{attribute 'GeneratedUsingTerminal: EL6631-0000-0018'}
{attribute addProperty BoxType "EL6631-0000-0018"}
{attribute addProperty Id "AdsAddrAT %I*TcoIo.TcoAmsAddr0AoeNetIdAT %I*TcoIo.TcoAmsNetId0StateAT %I*UINT2"}
{attribute addProperty CRC "2407881067"}
{attribute addProperty Size "2"}
TYPE InfoData_8F85596B EXTENDS TcoIo.InputBase_8311D824 :
STRUCT
	{attribute addProperty Name "AdsAddr"}
	AdsAddr AT %I* : TcoIo.TcoAmsAddr;
	{attribute addProperty Name "AoeNetId"}
	AoeNetId AT %I* : TcoIo.TcoAmsNetId;
	{attribute addProperty Name "State"}
	State AT %I* : UINT;
END_STRUCT
END_TYPE

(* stored: Version 1.2.0.0, ProductVersion 3.1.4024.11
   DUT InfoData_8F85596B: Id {1aa0af1e-65ef-0b9e-06db-f0f9f447082e} *)
